(* PLC project comp_new, Dassault Systèmes ControlBuild 2024x Refresh1 *)
(* stored: creationDateTime 2024-04-12T15:53:24-01:00 *)

FUNCTION_BLOCK apnew.comp_new


END_FUNCTION_BLOCK
